PROGRAM Main_Buffer
VAR
	
END_VAR

(* save data to database *)
//Buffer_Data();
//Buffer_IMU();

END_PROGRAM

(* stored: Version 1.1.0.1, ProductVersion 3.1.4024.6
   POU Main_Buffer: Id {d634cea7-0b2b-4450-a767-f61c97526782}, SpecialFunc None *)
